Universal Robots PolyScope program: d_str.urp

Program d_str (installation=ext_control directory=/programs createdIn=5.17.3 lastSavedIn=5.17.3 robotSerialNumber=20245501435)
Calibrated DH parameters: a=[0.000154, -0.137004, -0.385524, -0.00002, 0.000092, 0]; d=[0.162441, 211.794786, -230.585024, 18.923638, 0.099786, 0.09951]; alpha=[1.569493, -0.001902, 0.003874, 1.570111, -1.570167, 0]; deltaTheta=[0, -1.242934, 1.056292, 0.186646, 0.000002, 0.000001]
InitVariablesNode
Robot Program (runOnlyOnce=false)
  MoveL speed 250 mm/s, acceleration 1200 mm/s^2 (useActiveTCP=true) feature=Joint_6_name
    Waypoint Waypoint_1: TCP in base x=256.548 y=665.973 z=108.569 mm, rx=-1.5374 ry=-2.2292 rz=1.2496 rad; joints [-127.734, -31.287, 72.205, -80.819, -83.87, -151.225] deg; TCP offset x=28.21 y=-96.107 z=-99.69 mm, rx=0 ry=0 rz=0 rad; feature pose in base x=256.557 y=665.972 z=108.574 mm, rx=-1.5375 ry=-2.2292 rz=1.2495 rad
    Waypoint Waypoint_2 (Relative): relativeFromPosition TCP in base x=256.565 y=665.975 z=108.582 mm, rx=-1.5375 ry=-2.2292 rz=1.2495 rad; joints [-127.735, -31.288, 72.203, -80.818, -83.87, -151.225] deg; TCP in base x=308.201 y=212.166 z=168.469 mm, rx=1.5669 ry=2.3637 rz=-1.3134 rad; joints [-170.092, -63.301, 129.774, -117.857, -124.063, -180.489] deg; feature pose in base x=308.201 y=212.166 z=168.469 mm, rx=1.5669 ry=2.3637 rz=-1.3134 rad
